(* CODESYS project IO.library
   Company: MyCompany DAFRA1
   DefaultNamespace: IO
   Version: 0.1.0.0
   Placeholder: IO
   Author: Dejan Rozic
   Description: Lib for IO modules
   Title: IO

Project tree, tasks and I/O mapping:
  libraries: Tc2_Standard, * (Beckhoff Automation GmbH); Tc2_System, * (Beckhoff Automation GmbH); Tc3_Module, * (Beckhoff Automation GmbH)
  DUTs/
  GVLs/
  POUs/
    Actuator/
    Sensor/
      function block FB_TEST [ST]
    program MAIN [ST]
  Version/
    global variables Global_Version
  VISUs/
*)

// Version/Global_Version
{attribute 'TcGenerated'}
{attribute 'no-analysis'}
{attribute 'linkalways'}
// This function has been automatically generated from the project information.
VAR_GLOBAL CONSTANT
	{attribute 'const_non_replaced'}
	stLibVersion_IO_ : ST_LibVersion := (iMajor := 0, iMinor := 1, iBuild := 0, iRevision := 0, nFlags := 0, sVersion := '0.1.0.0');
END_VAR

// POUs/Sensor/FB_TEST
FUNCTION_BLOCK FB_TEST EXTENDS FB_TcAlarm
VAR_INPUT
END_VAR
VAR_OUTPUT
END_VAR
VAR
	var1 : BOOL;
END_VAR

var1 := TRUE;

END_FUNCTION_BLOCK

// POUs/MAIN
PROGRAM MAIN
VAR
END_VAR

END_PROGRAM
